FUNCTION_BLOCK ChangeDetector (* Basic Function Block Type *)
  (* Standard: 61499-2 *)
  (* Version 0.0, 11/2/2016, chivdan, nxtControl GmbH, Template *)
  PACKAGE Main;
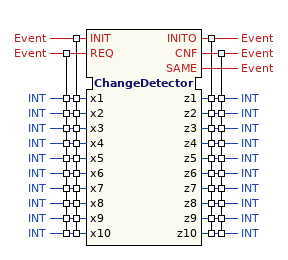
  EVENT_INPUT
    INIT WITH x1, x2, x3, x4, x5, x6, x7, x8, x9, x10;
    REQ WITH x1, x2, x3, x4, x5, x6, x7, x8, x9, x10; (* Normal Execution Request *)
  END_EVENT
  EVENT_OUTPUT
    INITO WITH z1, z2, z3, z4, z5, z6, z7, z8, z9, z10;
    CNF WITH z1, z2, z3, z4, z5, z6, z7, z8, z9, z10; (* Execution Confirmation *)
    SAME;
  END_EVENT
  VAR_INPUT
    x1 : INT; (* Input event qualifier *)
    x2 : INT;
    x3 : INT;
    x4 : INT;
    x5 : INT;
    x6 : INT;
    x7 : INT;
    x8 : INT;
    x9 : INT;
    x10 : INT;
  END_VAR
  VAR_OUTPUT
    z1 : INT; (* Output event qualifier *)
    z2 : INT;
    z3 : INT;
    z4 : INT;
    z5 : INT;
    z6 : INT;
    z7 : INT;
    z8 : INT;
    z9 : INT;
    z10 : INT;
  END_VAR
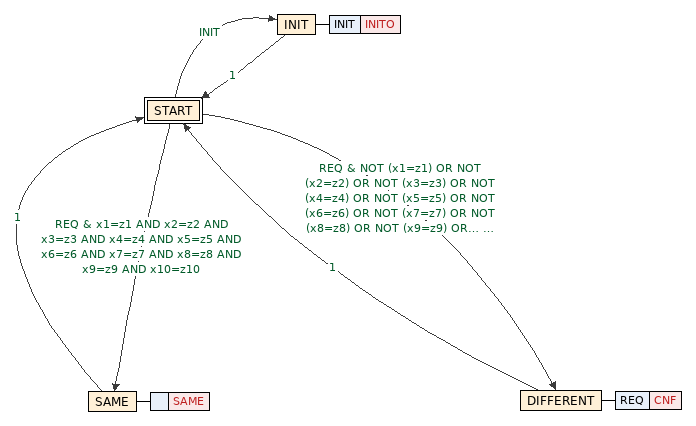
  EC_STATES
    START; (* Initial State *)
    INIT : INIT -> INITO; (* Initialization *)
    SAME : -> SAME; (* Normal execution *)
    DIFFERENT : REQ -> CNF;
  END_STATES
  EC_TRANSITIONS
    START TO INIT := INIT;
    INIT TO START := 1;
    START TO SAME := REQ & x1=z1 AND x2=z2 AND x3=z3 AND x4=z4 AND x5=z5 AND x6=z6 AND x7=z7 AND x8=z8 AND x9=z9 AND x10=z10;
    SAME TO START := 1;
    START TO DIFFERENT := REQ & NOT (x1=z1) OR NOT (x2=z2) OR NOT (x3=z3) OR NOT (x4=z4) OR NOT (x5=z5) OR NOT (x6=z6) OR NOT (x7=z7) OR NOT (x8=z8) OR NOT (x9=z9) OR NOT (x10=z10);
    DIFFERENT TO START := 1;
  END_TRANSITIONS
  ALGORITHM INIT IN ST: (* Initialization algorithm *)
;
z1:=0;
z2:=0;
z3:=0;
z4:=0;
z5:=0;
z6:=0;
z7:=0;
z8:=0;
z9:=0;
z10:=0;
  END_ALGORITHM
  ALGORITHM REQ IN ST: (* Normally executed algorithm *)
;
z1:=x1;
z2:=x2;
z3:=x3;
z4:=x4;
z5:=x5;
z6:=x6;
z7:=x7;
z8:=x8;
z9:=x9;
z10:=x10;
  END_ALGORITHM
END_FUNCTION_BLOCK
